(* PLC project cmd_motor_1d2s, Dassault Systèmes ControlBuild 2024x *)
(* stored: creationDateTime 2023-10-03T11:13:34-01:00 *)

FUNCTION_BLOCK actuator
  VAR_INPUT
    autoMode : BOOL := false;
    manualMode : BOOL := false;
  END_VAR
  VAR_INPUT
    autoHSCmd : BOOL := false;
    autoLSCmd : BOOL := false;
  END_VAR
  VAR_INPUT
    highSpeedPB : BOOL := false;
    lowSpeedPB : BOOL := false;
    stopPB : BOOL := false;
  END_VAR
  VAR_INPUT
    generalFault : BOOL := false;
  END_VAR
  VAR_OUTPUT
    highSpeedCmd : BOOL := false;
    lowSpeedCmd : BOOL := false;
  END_VAR

(* LD diagram, written out as Structured Text *)
1:
highSpeedCmd := (autoMode AND autoHSCmd OR manualMode AND (highSpeedPB OR highSpeedCmd) AND NOT lowSpeedPB AND NOT stopPB) AND NOT generalFault;
2:
lowSpeedCmd := (autoMode AND autoLSCmd OR manualMode AND (lowSpeedPB OR lowSpeedCmd) AND NOT highSpeedPB AND NOT stopPB) AND NOT generalFault;
END_FUNCTION_BLOCK

FUNCTION_BLOCK faults
  VAR_INPUT
    highSpeedCmd : BOOL := false;
    lowSpeedCmd : BOOL := false;
  END_VAR
  VAR_INPUT
    thermalFB : BOOL := false;
    highSpeedFB : BOOL := false;
    lowSpeedFB : BOOL := false;
  END_VAR
  VAR_INPUT
    acknowledgePB : BOOL := false;
  END_VAR
  VAR_OUTPUT
    generalFault : BOOL := false;
  END_VAR
  VAR
    thermalFault : BOOL := false;
    highSpeedFBFault : BOOL := false;
    lowSpeedFBFault : BOOL := false;
  END_VAR

(* LD diagram, written out as Structured Text *)
1:
IF acknowledgePB THEN thermalFault := FALSE; END_IF;
IF acknowledgePB THEN highSpeedFBFault := FALSE; END_IF;
IF acknowledgePB THEN lowSpeedFBFault := FALSE; END_IF;
IF acknowledgePB THEN generalFault := FALSE; END_IF;
2:
TON_HI(IN := highSpeedCmd, PT := T#0h0m2s0ms);
IF TON_HI.Q0 AND NOT highSpeedFB THEN highSpeedFBFault := TRUE; END_IF;
TON_LO(IN := lowSpeedCmd, PT := T#0h0m2s0ms);
IF TON_LO.Q0 AND NOT lowSpeedFB THEN lowSpeedFBFault := TRUE; END_IF;
3:
IF NOT thermalFB THEN thermalFault := TRUE; END_IF;
4:
IF thermalFault OR highSpeedFBFault OR lowSpeedFBFault THEN generalFault := TRUE; END_IF;
END_FUNCTION_BLOCK

(* Command of a motor with one direction and two speeds and with fault detection *)
PROGRAM cmd_equipment_library.cmd_motor_1d2s
  VAR_INPUT
    autoMode : BOOL := false;
    manualMode : BOOL := false;
  END_VAR
  VAR_INPUT
    autoHSCmd : BOOL := false;
    autoLSCmd : BOOL := false;
  END_VAR
  VAR_INPUT
    highSpeedPB : BOOL := false;
    lowSpeedPB : BOOL := false;
    stopPB : BOOL := false;
  END_VAR
  VAR_INPUT
    thermalFB : BOOL := false;
    highSpeedFB : BOOL := false;
    lowSpeedFB : BOOL := false;
  END_VAR
  VAR_INPUT
    acknowledgePB : BOOL := false;
  END_VAR
  VAR_OUTPUT
    highSpeedCmd : BOOL := false;
    lowSpeedCmd : BOOL := false;
  END_VAR
  VAR_OUTPUT
    generalFault : BOOL := false;
  END_VAR

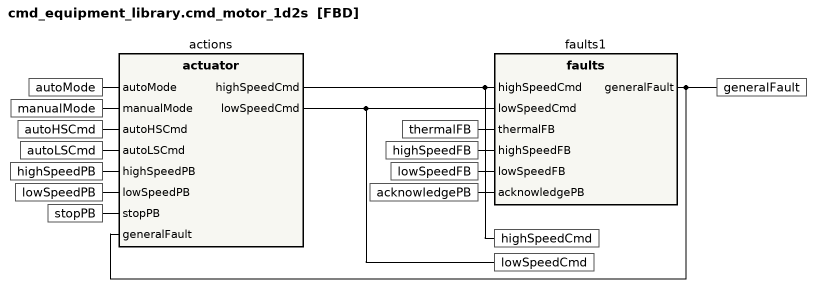
(* FBD diagram, written out as Structured Text *)
faults1(highSpeedCmd := actions.highSpeedCmd, lowSpeedCmd := actions.lowSpeedCmd, thermalFB := thermalFB, highSpeedFB := highSpeedFB, lowSpeedFB := lowSpeedFB, acknowledgePB := acknowledgePB);
actions(autoMode := autoMode, manualMode := manualMode, autoHSCmd := autoHSCmd, autoLSCmd := autoLSCmd, highSpeedPB := highSpeedPB, lowSpeedPB := lowSpeedPB, stopPB := stopPB, generalFault := faults1.generalFault);
highSpeedCmd := actions.highSpeedCmd;
lowSpeedCmd := actions.lowSpeedCmd;
generalFault := faults1.generalFault;
END_PROGRAM
